// TIA Portal V17 export
// export: Created 2024-06-19T09:47:09.9765736Z, ExportSetting WithDefaults, DisplayName Totally Integrated Automation Portal, DisplayVersion V17, DisplayName TIA Portal Openness, DisplayVersion V17, DisplayName TIA Portal Version Control Interface, DisplayVersion V17, DisplayName STEP 7 Professional, DisplayVersion V17, DisplayName STEP 7 Safety, DisplayVersion V17, DisplayName WinCC Professional, DisplayVersion V17
ORGANIZATION_BLOCK "Main"   // OB1, LAD, ProgramCycle
TITLE = "Main Program Sweep (Cycle)"
{ S7_Optimized_Access := 'TRUE' }
VERSION : 0.1
// *********************  Création : 01/06/2024  *********************
// *****************  Kep Technologies - Caluire 69150  ****************
// ************************  RM Automation  ***********************
// **********************  Auteur: Rebouh.M  ***********************
// ***************** Contact : Rebouh.mehdi@hotmail.fr  ***************
// stored: AutoNumber true, IsIECCheckEnabled false, SetENOAutomatically false
   VAR_INPUT
      Initial_Call : Bool;   // Initial call of this OB
      Remanence : Bool;   // =True, if remanent data are available
   END_VAR
BEGIN

REGION Network 1: Manager
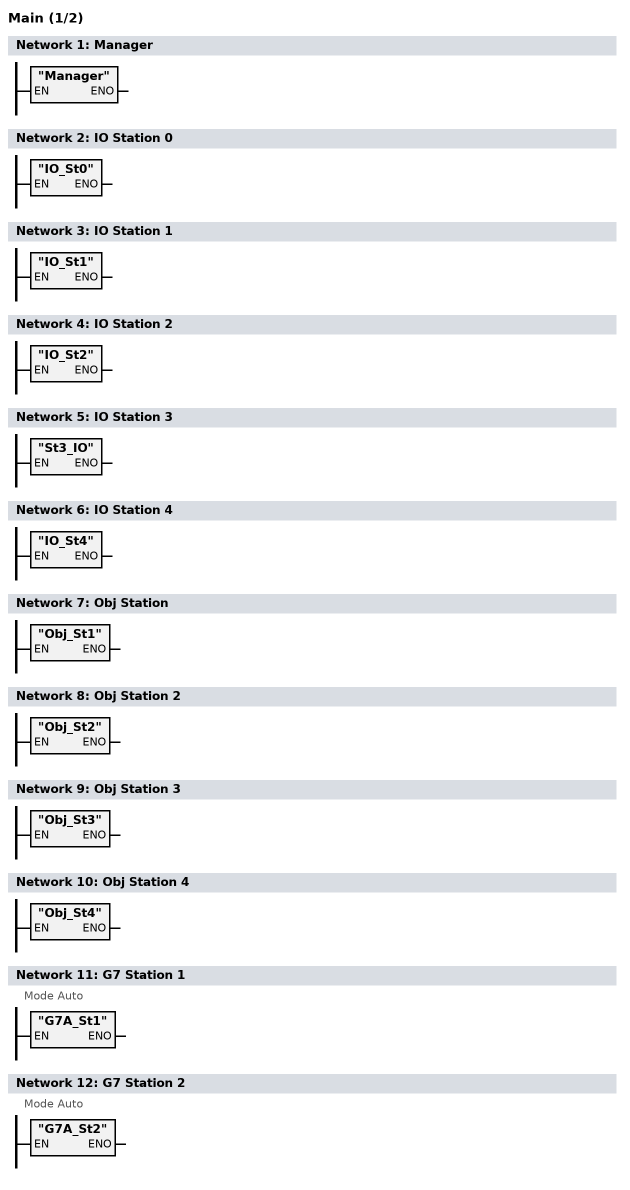
   RUNG wire#powerrail
      "Manager"()
   END_RUNG
   // the same network as SCL:
   "Manager"();
END_REGION

REGION Network 2: IO Station 0
   RUNG wire#powerrail
      "IO_St0"()
   END_RUNG
   // the same network as SCL:
   "IO_St0"();
END_REGION

REGION Network 3: IO Station 1
   RUNG wire#powerrail
      "IO_St1"()
   END_RUNG
   // the same network as SCL:
   "IO_St1"();
END_REGION

REGION Network 4: IO Station 2
   RUNG wire#powerrail
      "IO_St2"()
   END_RUNG
   // the same network as SCL:
   "IO_St2"();
END_REGION

REGION Network 5: IO Station 3
   RUNG wire#powerrail
      "St3_IO"()
   END_RUNG
   // the same network as SCL:
   "St3_IO"();
END_REGION

REGION Network 6: IO Station 4
   RUNG wire#powerrail
      "IO_St4"()
   END_RUNG
   // the same network as SCL:
   "IO_St4"();
END_REGION

REGION Network 7: Obj Station
   RUNG wire#powerrail
      "Obj_St1"()
   END_RUNG
   // the same network as SCL:
   "Obj_St1"();
END_REGION

REGION Network 8: Obj Station 2
   RUNG wire#powerrail
      "Obj_St2"()
   END_RUNG
   // the same network as SCL:
   "Obj_St2"();
END_REGION

REGION Network 9: Obj Station 3
   RUNG wire#powerrail
      "Obj_St3"()
   END_RUNG
   // the same network as SCL:
   "Obj_St3"();
END_REGION

REGION Network 10: Obj Station 4
   RUNG wire#powerrail
      "Obj_St4"()
   END_RUNG
   // the same network as SCL:
   "Obj_St4"();
END_REGION

REGION Network 11: G7 Station 1
   // Mode Auto
   RUNG wire#powerrail
      "G7A_St1"()
   END_RUNG
   // the same network as SCL:
   "G7A_St1"();
END_REGION

REGION Network 12: G7 Station 2
   // Mode Auto
   RUNG wire#powerrail
      "G7A_St2"()
   END_RUNG
   // the same network as SCL:
   "G7A_St2"();
END_REGION

REGION Network 13: G7 Station 3
   // Mode Auto
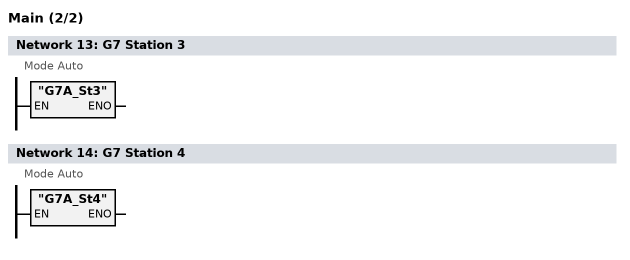
   RUNG wire#powerrail
      "G7A_St3"()
   END_RUNG
   // the same network as SCL:
   "G7A_St3"();
END_REGION

REGION Network 14: G7 Station 4
   // Mode Auto
   RUNG wire#powerrail
      "G7A_St4"()
   END_RUNG
   // the same network as SCL:
   "G7A_St4"();
END_REGION
END_ORGANIZATION_BLOCK
